// SIMATIC S7-200 SMART project (STEP 7-Micro/WIN SMART), CPU SR40

SYMBOL_TABLE 系统符号
Always_On        SM0.0    // 始终接通
Clock_1s         SM0.5    // 针对 1 s 的周期时间，时钟脉冲接通 0.5 s，断开 0.5 s.
END_SYMBOL_TABLE

ORGANIZATION_BLOCK MAIN:OB1
TITLE=程序注释
BEGIN
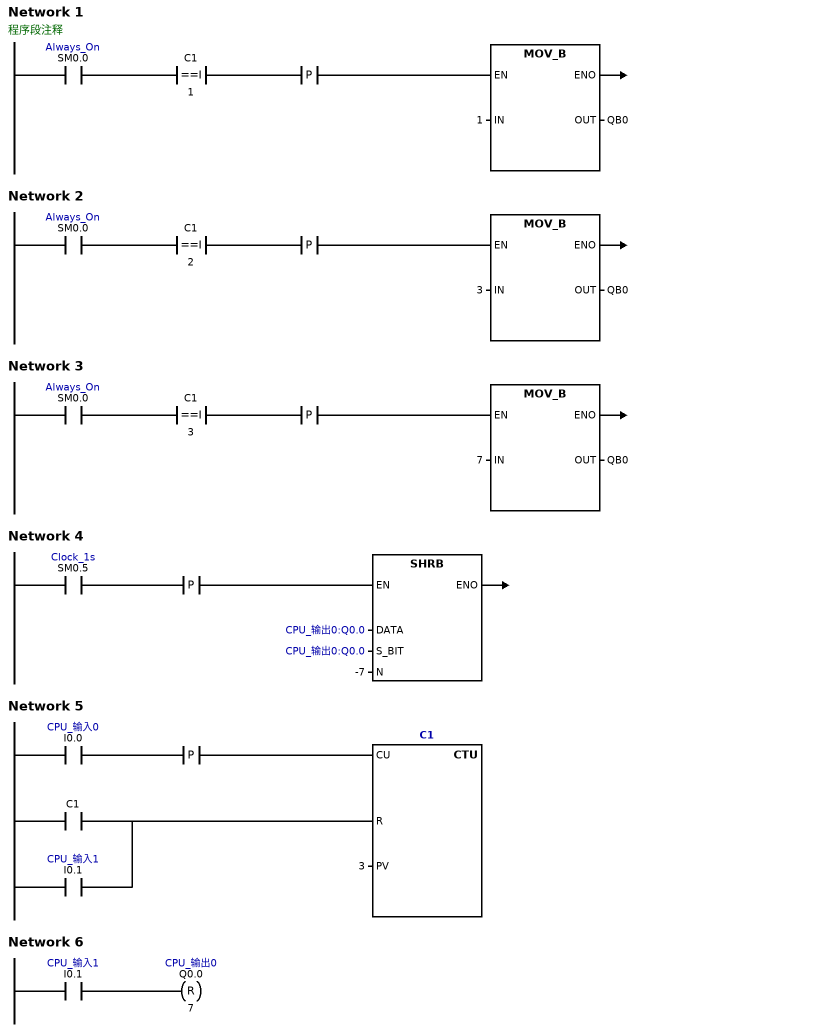
Network 1
// 程序段注释
LD     Always_On:SM0.0
AW=    C1, 1
EU
MOVB   1, QB0
Network 2
LD     Always_On:SM0.0
AW=    C1, 2
EU
MOVB   3, QB0
Network 3
LD     Always_On:SM0.0
AW=    C1, 3
EU
MOVB   7, QB0
Network 4
LD     Clock_1s:SM0.5
EU
SHRB   CPU_输出0:Q0.0, CPU_输出0:Q0.0, -7
Network 5
LD     CPU_输入0:I0.0
EU
LD     C1
O      CPU_输入1:I0.1
CTU    C1, 3
Network 6
// (network saved uncompiled; LAD cells follow)
// row 0: c0 -| |- CPU_输入1:I0.1  c1 -(R) CPU_输出0:Q0.0, 7
END_ORGANIZATION_BLOCK
